// TIA Portal V20 export
DATA_BLOCK "DB_DigitalInputsSonplas"   // DB2211
// stored: AutoNumber false, InstanceOfName FB_DigitalInputsSonplas, InstanceOfType FB
"FB_DigitalInputsSonplas"
   // VAR
   //    sSonplasDiagDPCoupler { S7_SetPoint := 'True'} : "FB_DigitalInput";
   //    sSonplasReady { S7_SetPoint := 'True'} : "FB_DigitalInput";
   //    sSonplasNoEStop { S7_SetPoint := 'True'} : "FB_DigitalInput";
   //    sSonplasDoorsClosed { S7_SetPoint := 'True'} : "FB_DigitalInput";
   //    sSonplasRunError { S7_SetPoint := 'True'} : "FB_DigitalInput";
   //    sSonplasFreeI200_5 { S7_SetPoint := 'True'} : "FB_DigitalInput";
   //    sSonplasFreeI200_6 { S7_SetPoint := 'True'} : "FB_DigitalInput";
   //    sSonplasFreeI200_7 { S7_SetPoint := 'True'} : "FB_DigitalInput";
   //    sSonplasFreeI201_0 { S7_SetPoint := 'True'} : "FB_DigitalInput";
   //    sSonplasOutCollision { S7_SetPoint := 'True'} : "FB_DigitalInput";
   //    sSonplasFreeI201_2 { S7_SetPoint := 'True'} : "FB_DigitalInput";
   //    Sonpla_FreeI201_3 { S7_SetPoint := 'True'} : "FB_DigitalInput";
   //    sSonplasFreeI201_4 { S7_SetPoint := 'True'} : "FB_DigitalInput";
   //    sSonplasFreeI201_5 { S7_SetPoint := 'True'} : "FB_DigitalInput";
   //    sSonplasFreeI201_6 { S7_SetPoint := 'True'} : "FB_DigitalInput";
   //    sSonplasFreeI201_7 { S7_SetPoint := 'True'} : "FB_DigitalInput";
   //    sSonplasShuttle1Finished { S7_SetPoint := 'True'} : "FB_DigitalInput";
   //    sSonplasFreeI202_1 { S7_SetPoint := 'True'} : "FB_DigitalInput";
   //    sSonplasFreeI202_2 { S7_SetPoint := 'True'} : "FB_DigitalInput";
   //    sSonplasFreeI202_3 { S7_SetPoint := 'True'} : "FB_DigitalInput";
   //    sSonplasFreeI202_4 { S7_SetPoint := 'True'} : "FB_DigitalInput";
   //    sSonplasFreeI202_5 { S7_SetPoint := 'True'} : "FB_DigitalInput";
   //    sSonplasFreeI202_6 { S7_SetPoint := 'True'} : "FB_DigitalInput";
   //    sSonplasFreeI202_7 { S7_SetPoint := 'True'} : "FB_DigitalInput";
   //    sSonplasShuttle2Finished { S7_SetPoint := 'True'} : "FB_DigitalInput";
   //    sSonplasFreeI203_1 { S7_SetPoint := 'True'} : "FB_DigitalInput";
   //    sSonplasFreeI203_2 { S7_SetPoint := 'True'} : "FB_DigitalInput";
   //    sSonplasFreeI203_3 { S7_SetPoint := 'True'} : "FB_DigitalInput";
   //    sSonplasFreeI203_4 { S7_SetPoint := 'True'} : "FB_DigitalInput";
   //    sSonplasFreeI203_5 { S7_SetPoint := 'True'} : "FB_DigitalInput";
   //    sSonplasFreeI203_6 { S7_SetPoint := 'True'} : "FB_DigitalInput";
   //    sSonplasFreeI203_7 { S7_SetPoint := 'True'} : "FB_DigitalInput";
   //    sSonplasFlowResultAvail { S7_SetPoint := 'True'} : "FB_DigitalInput";
   //    sSonplasFreeI244_1 { S7_SetPoint := 'True'} : "FB_DigitalInput";
   //    sSonplasFreeI244_2 { S7_SetPoint := 'True'} : "FB_DigitalInput";
   //    sSonplasFreeI244_3 { S7_SetPoint := 'True'} : "FB_DigitalInput";
   //    sSonplasFreeI244_4 { S7_SetPoint := 'True'} : "FB_DigitalInput";
   //    sSonplasFreeI244_5 { S7_SetPoint := 'True'} : "FB_DigitalInput";
   //    sSonplasFreeI244_6 { S7_SetPoint := 'True'} : "FB_DigitalInput";
   //    sSonplasFreeI244_7 { S7_SetPoint := 'True'} : "FB_DigitalInput";
   // END_VAR
BEGIN
END_DATA_BLOCK
